TYPE Astrofan612FfuLoopConfig :
STRUCT
	IsEnabled : BOOL;
	FfuLoopStandardSetSpeed : UINT;
	FfuLoopPressureTimerSeconds : UINT;
	FfuLoopWarning 	: Astrofan612FfuEvent;
	FfuLoopAlarm 	: Astrofan612FfuEvent;
	FfuPressureMinimumValuePa : UINT;
	FfuPressureMaximumValuePa : UINT;
	FfuLoopSetSpeedHigherLimitPercent : UINT;
	FfuLoopSetSpeedLowerLimitPercent : UINT;
END_STRUCT
END_TYPE

(* stored: Version 1.1.0.1, ProductVersion 3.1.4024.12
   DUT Astrofan612FfuLoopConfig: Id {e7d80be7-83de-4318-9524-5326bbf4c589} *)
